// TIA Portal V21 export
DATA_BLOCK "ProcessAlarms"   // DB191
{ S7_Optimized_Access := 'FALSE' }
// stored: AutoNumber false
   VAR
      CipCycleOver : Bool;
      CipCycleConductivityReached : Bool;
      CipCycleConductivityNotReached : Bool;
      ConductivityNotSampled : Bool;
      CipReportDataNotLogged : Bool;
      PhtFailed : Bool;
      PhtPassed : Bool;
      PhtOver : Bool;
      PhtReportDataNotLogged : Bool;
      SterilizationTimeOver : Bool;
      SteamFlowLow : Bool;
      SterilizationHighTemperature : Bool;
      SterilizationCycleCompleted : Bool;
      SterilizationReportDataNotLogged : Bool;
      WfiFlowLow : Bool;
      BatchWfiFlowLow : Bool;
   END_VAR
BEGIN
END_DATA_BLOCK
